RoboDK station: MergePrograms.rdk

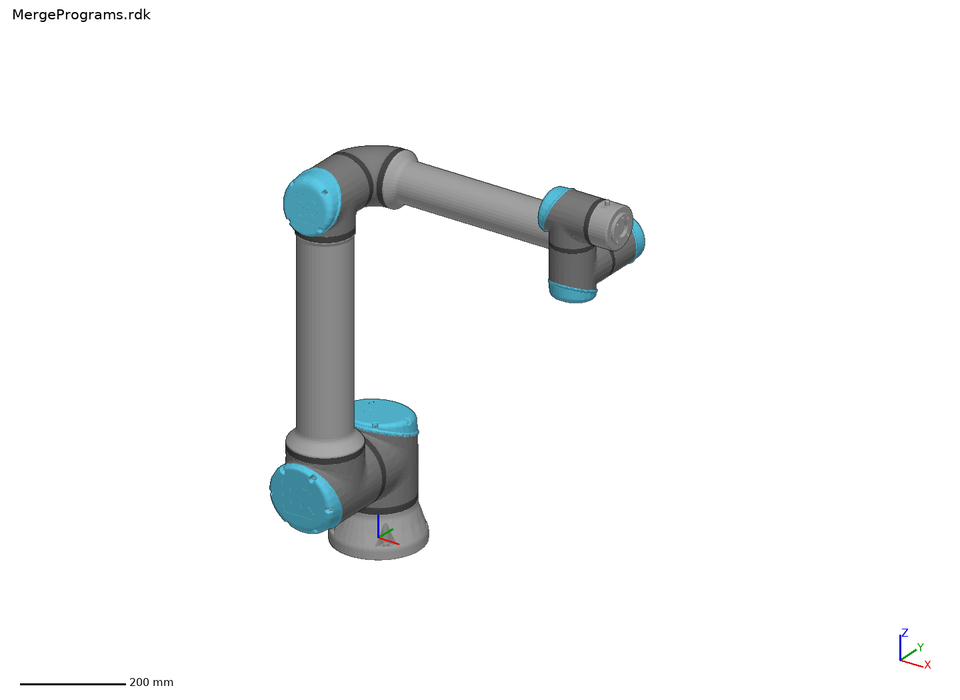
[picture v0: the station drawn from its stored meshes, robots at their saved joint values, targets as dots, program paths as lines]
Station MergePrograms (saved by RoboDK 5.5.2). Poses are relative to the parent item; angles as X-Y-Z fixed-axis rotations.
  - frame UR10e Base at (0, 1000, 0) mm
    - robot UR10e: 6 axes, payload 10 kg, reach 1300 mm, repeatability 0.05 mm, weight 28.9 kg
        modified DH rows (alpha deg, a mm, theta deg, d mm): 0, 0, 0, 180.7; 90, 0, 180, 0; 0, 612.6, 0, 0; 0, 571.335, 0, 174.15; -90, 0, 0, 119.85; 90, 0, 180, 116.55
        joint limits [-360, -360, -360, -360, -360, -360] to [360, 360, 360, 360, 360, 360]; home [0, -90, -90, 0, 90, 0]; saved at [0, -90, -90, 0, 90, 0]
  - program Prog1 (2 instructions, listed below)
  - program Prog2 (2 instructions, listed below)
  - program Prog3 (1 instructions, listed below)
  - program Prog1 Prog2 Prog3 Merged (5 instructions, listed below)

--- program Prog1 (robot UR10e) ---
  Print: Prog1
  Call Prog2

--- program Prog2 (robot UR10e) ---
  Print: Prog2
  Call Prog3

--- program Prog3 (robot UR10e) ---
  Print: Prog3

--- program Prog1 Prog2 Prog3 Merged (robot UR10e) ---
  Print: Prog1
  Call Prog2
  Print: Prog2
  Call Prog3
  Print: Prog3
